FUNCTION F_GetElementInterface : ST_ElementInterface
(**************************************************************************************
 * 	Application		:	BoxControl Framework
 *	Revision		:	$Revision: 404529 $
 *	Revision date	:	$Date: 2018-04-23 08:21:38 +0200 (Mo., 23 Apr 2018) $
 *	Last changed by	:	$Author: b7bolm $
 *	URL				:	$URL: http://almscdc.swisslog.com/repo/SWPD/Development/BoxControlFramework/20_Release/trunk/01_Software/BCF/BCF/JumpStart/20_Product/10_App/13_Elements/10_Lib/10_Conv/10_Functions/F_GetElementInterface.TcPOU $
 *
 *	Purpose			:	Returns element interface
 *
 * ------------------------------------------------------------------------------------
 *	Copyright Swisslog [IP AG], Switzerland. All rights reserved.
 * 
 * ------------------------------------------------------------------------------------
 *	
 * 	Revision History: 
 *
 * 	VERSION			DATE			INITIALS			DESCRIPTION
 *	0.1				01.01.2001		swl					Example
 *
 **************************************************************************************)
VAR_INPUT
	eElementNumber		: E_ElementNumber;
END_VAR


// Check if function number is valid
IF eElementNumber > E_ElementNumber.E_BEGIN_ELEMENT AND
   eElementNumber < E_ElementNumber.E_END_ELEMENT THEN
	
   // Check reference is valid
   IF __ISVALIDREF(ElementRegistry[eElementNumber].rElement) THEN
	   
   		// Return element interface
   		F_GetElementInterface := ElementRegistry[eElementNumber].rElementInterface;
   END_IF
END_IF

END_FUNCTION

(* stored: Version 1.1.0.1, ProductVersion 3.1.4022.12
   POU F_GetElementInterface: Id {6f84afa5-81a4-410d-90e3-a9ab6eac45ea}, SpecialFunc None *)
